// TIA Portal V17 export
// export: Created 2024-09-02T12:50:04.1377322Z, ExportSetting WithDefaults, DisplayName Totally Integrated Automation Portal, DisplayVersion V17, DisplayName TIA Portal Openness, DisplayVersion V17, DisplayName TIA Portal Version Control Interface, DisplayVersion V17, DisplayName STEP 7 Professional, DisplayVersion V17, DisplayName STEP 7 Safety, DisplayVersion V17, DisplayName WinCC Professional, DisplayVersion V17
FUNCTION_BLOCK "SysFB_RF300"   // FB809, LAD
TITLE = /RF300 Read / Write / RF300 Lesen / Schreiben
{ S7_Optimized_Access := 'TRUE' }
AUTHOR : STEAM
FAMILY : MOBY
NAME : MOBY
VERSION : 0.1
// stored: AutoNumber true, IsIECCheckEnabled false, IsRetainMemResEnabled false, MemoryReserve 100, SetENOAutomatically false, UDAEnableTagReadback false
   VAR_INPUT
      HW_ID : Int;   // Hardware ID
      HW_ADR : Int;   // Hardwareadresse / Hardware address
      Channel : Int;   // Kanalnummer (1..2) / Channel number (1..2)
      RF_Type : Bool;   // False=RF300 True= RF200
      "Fault ACK" : Bool;   // Fehler quittieren / Acknowledge error
      "New Start" : Bool;   // Flanke Neustart / Flank Restart
   END_VAR
   VAR_OUTPUT
      Fault : Bool;   // es ist ein Fehler aufgetreten / An error has occurred.
      "MDS Present" : Bool;   // Datenträger ist anwesend / Data carrier is present
      HMIDiag : "TypeMobyHMIDiag";   // HMI Diagnose / HMI Diagnosis
   END_VAR
   VAR_IN_OUT
      Command : "TypeMobyBefehle";
   END_VAR
   VAR
      hwConnect { S7_SetPoint := 'True'} : IID_HW_CONNECT;
      Reset : Struct
         Start : Bool;   // Start
         Active : Bool;   // Aktiv / Active
         Finish : Bool;   // Fertig / Finished
         Fault : Bool;   // Fehler / Error
         Status : DWord;   // Status
         Status_marked : DWord;   // Status
         Num_Of_OK : DInt;   // Anzahl IO / Number NIO
         Num_Of_NOK : DInt;   // Anzahl NIO / Number NIO
         started : Bool;   // Funktion gestartet / Function started
         fp_started : Bool;   // flanke gestartet / Flank started
         hm_fp_started : Bool;   // HM flanke gestartet / HM flank started
         Finish_OK : Bool;   // Fertig IO / Finish IO
         fp_Finish_OK : Bool;   // flanke Fertig IO / Flank finished OK
         "hm fp_Finish_OK" : Bool;   // hm flanke Fertig IO / hm flank finished IO
         Finish_NOK : Bool;   // Fertig NIO / Finish NIO
         fp_Finish_NOK : Bool;   // flanke Fertig IO / Flank finished OK
         "hm fp_Finish_NOK" : Bool;   // hm flanke Fertig IO / hm flank finished IO
         RunningTime : Time;
      END_STRUCT;
      Read : Struct
         Start : Bool;   // Start
         Active : Bool;   // Aktiv / Active
         Finish : Bool;   // Fertig / Finished
         Faul : Bool;   // Fehler / Error
         MDS_present : Bool;   // Datenträger vorhanden / Data carrier available
         Status : DWord;   // Status
         Status_marked : DWord;   // Status
         Num_Of_OK : DInt;   // Anzahl IO / Number NIO
         Num_Of_NOK : DInt;   // Anzahl NIO / Number NIO
         started : Bool;   // Funktion gestartet / Function started
         fp_started : Bool;   // flanke gestartet / Flank started
         hm_fp_started : Bool;   // HM flanke gestartet / HM flank started
         Finish_OK : Bool;   // Fertig IO / Finish IO
         fp_Finish_OK : Bool;   // flanke Fertig IO / Flank finished OK
         "hm fp_Finish_OK" : Bool;   // hm flanke Fertig IO / hm flank finished IO
         Finish_NOK : Bool;   // Fertig NIO / Finish NIO
         fp_Finish_NOK : Bool;   // flanke Fertig IO / Flank finished OK
         "hm fp_Finish_NOK" : Bool;   // hm flanke Fertig IO / hm flank finished IO
         RunningTime : Time;
      END_STRUCT;
      Write : Struct
         Start : Bool;   // Start
         Active : Bool;   // Aktiv / Active
         Finish : Bool;   // Fertig / Finished
         Fault : Bool;   // Fehler / Error
         MDS_present : Bool;   // Datenträger vorhanden / Data carrier available
         Status : DWord;   // Status
         Status_marked : DWord;   // Status
         Num_Of_OK : DInt;   // Anzahl IO / Number NIO
         Num_Of_NOK : DInt;   // Anzahl NIO / Number NIO
         started : Bool;   // Funktion gestartet / Function started
         fp_started : Bool;   // flanke gestartet / Flank started
         hm_fp_started : Bool;   // HM flanke gestartet / HM flank started
         Finish_OK : Bool;   // Fertig IO / Finish IO
         fp_Finish_OK : Bool;   // flanke Fertig IO / Flank finished OK
         "hm fp_Finish_OK" : Bool;   // hm flanke Fertig IO / hm flank finished IO
         Finish_NOK : Bool;   // Fertig NIO / Finish NIO
         fp_Finish_NOK : Bool;   // flanke Fertig IO / Flank finished OK
         "hm fp_Finish_NOK" : Bool;   // hm flanke Fertig IO / hm flank finished IO
         RunningTime : Time;
      END_STRUCT;
      SysDI_Reset { S7_SetPoint := 'True'} : Reset_RF300;
      SysDI_Read { S7_SetPoint := 'True'} : Read;
      SysDI_Write { S7_SetPoint := 'True'} : Write;
      SystemTime : Time;
      SystemTime_Old : Time;
      CycleTime : Time;
      ReadData : Struct
         SequenceNr : Int;
         RetVal : Word;
         Pos : DInt;
         finish : Bool;
      END_STRUCT;
      WriteData : Struct
         SequenceNr : Int;
         RetVal : Word;
         Pos : DInt;
         finish : Bool;
      END_STRUCT;
      ConnectionCheck : Struct
         TimeWithoutAction : Time;
         start : Bool;
         fp_start : Bool;
         HM_fp_start : Bool;
      END_STRUCT;
      "Checking Faults" : Struct
         FaultOccured : Bool;
         fp_FaultOccured : Bool;
         HM_fp_FaultOccured : Bool;
         TimeoutFault : Bool;
      END_STRUCT;
      SysDI_Reset200 { S7_SetPoint := 'True'} : Reset_RF200;
   END_VAR
   VAR_TEMP
      t_VKE0 : Bool;
      t_VKE1 : Bool;
      t_End : Bool;
      t_RF300_Ready : Bool;
      t_Befehl_INIT : "TypeMobySequenz";
   END_VAR
   VAR_TEMP   // added for the SCL form of the ladder/FBD networks
      _w1 : Bool;
      _w2 : Bool;
      _w3 : Bool;
   END_VAR
BEGIN

REGION Network 1: INIT
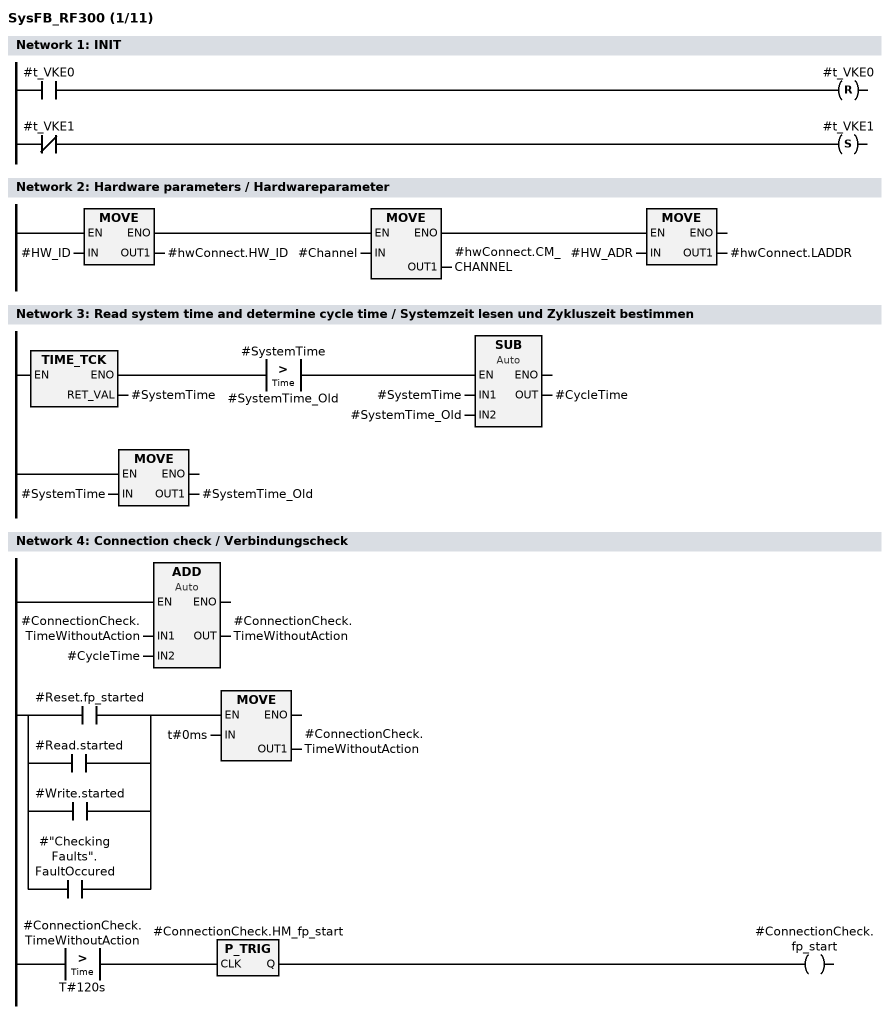
   RUNG wire#powerrail
      Contact( #t_VKE0 )
      R_Coil( #t_VKE0 )
   END_RUNG
   RUNG wire#powerrail
      I_Contact( #t_VKE1 )
      S_Coil( #t_VKE1 )
   END_RUNG
   // the same network as SCL:
   IF #t_VKE0 THEN #t_VKE0 := FALSE; END_IF;
   IF NOT #t_VKE1 THEN #t_VKE1 := TRUE; END_IF;
END_REGION

REGION Network 2: Hardware parameters / Hardwareparameter
   RUNG wire#powerrail
      Move(in := #HW_ID, out1 => #hwConnect.HW_ID)
      Move(in := #Channel, out1 => #hwConnect.CM_CHANNEL)
      Move(in := #HW_ADR, out1 => #hwConnect.LADDR)
   END_RUNG
   // the same network as SCL:
   #hwConnect.HW_ID := #HW_ID;
   #hwConnect.CM_CHANNEL := #Channel;
   #hwConnect.LADDR := #HW_ADR;
END_REGION

REGION Network 3: Read system time and determine cycle time / Systemzeit lesen und Zykluszeit bestimmen
   RUNG wire#powerrail
      TIME_TCK(RET_VAL => #SystemTime)
      { S7_Templates := "SrcType := Time" } GT_Contact(in1 := #SystemTime, in2 := #SystemTime_Old)
      Sub(in1 := #SystemTime, in2 := #SystemTime_Old, out => #CycleTime)
   END_RUNG
   RUNG wire#powerrail
      Move(in := #SystemTime, out1 => #SystemTime_Old)
   END_RUNG
   // the same network as SCL:
   #SystemTime := TIME_TCK(ENO => #_w1);
   IF #_w1 AND (#SystemTime > #SystemTime_Old) THEN #CycleTime := #SystemTime - #SystemTime_Old; END_IF;
   #SystemTime_Old := #SystemTime;
END_REGION

REGION Network 4: Connection check / Verbindungscheck
   RUNG wire#powerrail
      Add(in1 := #ConnectionCheck.TimeWithoutAction, in2 := #CycleTime, out => #ConnectionCheck.TimeWithoutAction)
   END_RUNG
   RUNG wire#powerrail
      Contact( #Reset.fp_started )
      wire#w1
      Move(in := t#0ms, out1 => #ConnectionCheck.TimeWithoutAction)
   END_RUNG
   RUNG wire#powerrail
      Contact( #Read.started )
   END_RUNG wire#w1
   RUNG wire#powerrail
      Contact( #Write.started )
   END_RUNG wire#w1
   RUNG wire#powerrail
      Contact( #"Checking Faults".FaultOccured )
   END_RUNG wire#w1
   RUNG wire#powerrail
      { S7_Templates := "SrcType := Time" } GT_Contact(in1 := #ConnectionCheck.TimeWithoutAction, in2 := T#120s)
      P_Trig( #ConnectionCheck.HM_fp_start )
      Coil( #ConnectionCheck.fp_start )
   END_RUNG
   // the same network as SCL:
   #ConnectionCheck.TimeWithoutAction := #ConnectionCheck.TimeWithoutAction + #CycleTime;
   IF #Reset.fp_started OR #Read.started OR #Write.started OR #"Checking Faults".FaultOccured THEN
       #ConnectionCheck.TimeWithoutAction := t#0ms;
   END_IF;
   #_w1 := #ConnectionCheck.TimeWithoutAction > T#120s;
   #_w2 := #_w1 AND NOT #ConnectionCheck.HM_fp_start;   // rising edge
   #ConnectionCheck.HM_fp_start := #_w1;
   #ConnectionCheck.fp_start := #_w2;
END_REGION

REGION Network 5: Error present / Fehler vorhanden
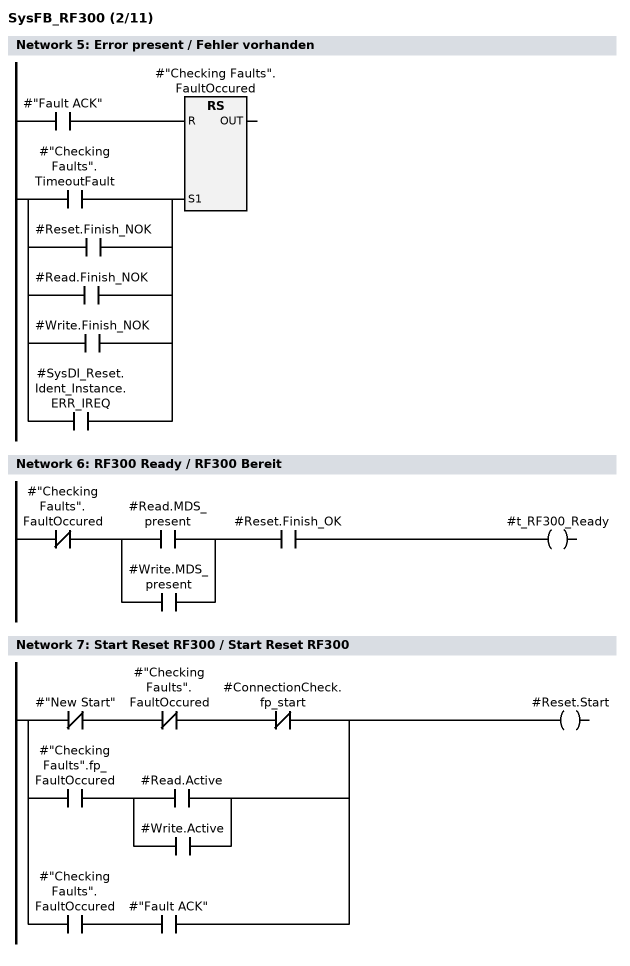
   RUNG wire#powerrail
      Contact( #"Fault ACK" )
      S_RS(operand := #"Checking Faults".FaultOccured, s1 := wire#w1)
   END_RUNG
   RUNG wire#powerrail
      Contact( #"Checking Faults".TimeoutFault )
   END_RUNG wire#w1
   RUNG wire#powerrail
      Contact( #Reset.Finish_NOK )
   END_RUNG wire#w1
   RUNG wire#powerrail
      Contact( #Read.Finish_NOK )
   END_RUNG wire#w1
   RUNG wire#powerrail
      Contact( #Write.Finish_NOK )
   END_RUNG wire#w1
   RUNG wire#powerrail
      Contact( #SysDI_Reset.Ident_Instance.ERR_IREQ )
   END_RUNG wire#w1
   // the same network as SCL:
   IF #"Fault ACK" THEN
       #"Checking Faults".FaultOccured := FALSE;   // RS flip-flop
   END_IF;
   IF #"Checking Faults".TimeoutFault OR #Reset.Finish_NOK OR #Read.Finish_NOK OR #Write.Finish_NOK OR #SysDI_Reset.Ident_Instance.ERR_IREQ THEN
       #"Checking Faults".FaultOccured := TRUE;
   END_IF;
END_REGION

REGION Network 6: RF300 Ready / RF300 Bereit
   RUNG wire#powerrail
      I_Contact( #"Checking Faults".FaultOccured )
      wire#w1
      Contact( #Read.MDS_present )
      wire#w2
      Contact( #Reset.Finish_OK )
      Coil( #t_RF300_Ready )
   END_RUNG
   RUNG wire#w1
      Contact( #Write.MDS_present )
   END_RUNG wire#w2
   // the same network as SCL:
   #t_RF300_Ready := NOT #"Checking Faults".FaultOccured AND (#Read.MDS_present OR #Write.MDS_present) AND #Reset.Finish_OK;
END_REGION

REGION Network 7: Start Reset RF300 / Start Reset RF300
   RUNG wire#powerrail
      I_Contact( #"New Start" )
      I_Contact( #"Checking Faults".FaultOccured )
      I_Contact( #ConnectionCheck.fp_start )
      wire#w1
      Coil( #Reset.Start )
   END_RUNG
   RUNG wire#powerrail
      Contact( #"Checking Faults".fp_FaultOccured )
      wire#w2
      Contact( #Read.Active )
   END_RUNG wire#w1
   RUNG wire#w2
      Contact( #Write.Active )
   END_RUNG wire#w1
   RUNG wire#powerrail
      Contact( #"Checking Faults".FaultOccured )
      Contact( #"Fault ACK" )
   END_RUNG wire#w1
   // the same network as SCL:
   #Reset.Start := (NOT #"New Start" AND NOT #"Checking Faults".FaultOccured AND NOT #ConnectionCheck.fp_start) OR (#"Checking Faults".fp_FaultOccured AND (#Read.Active OR #Write.Active)) OR (#"Checking Faults".FaultOccured AND #"Fault ACK");
END_REGION

REGION Network 8: Reset RF300
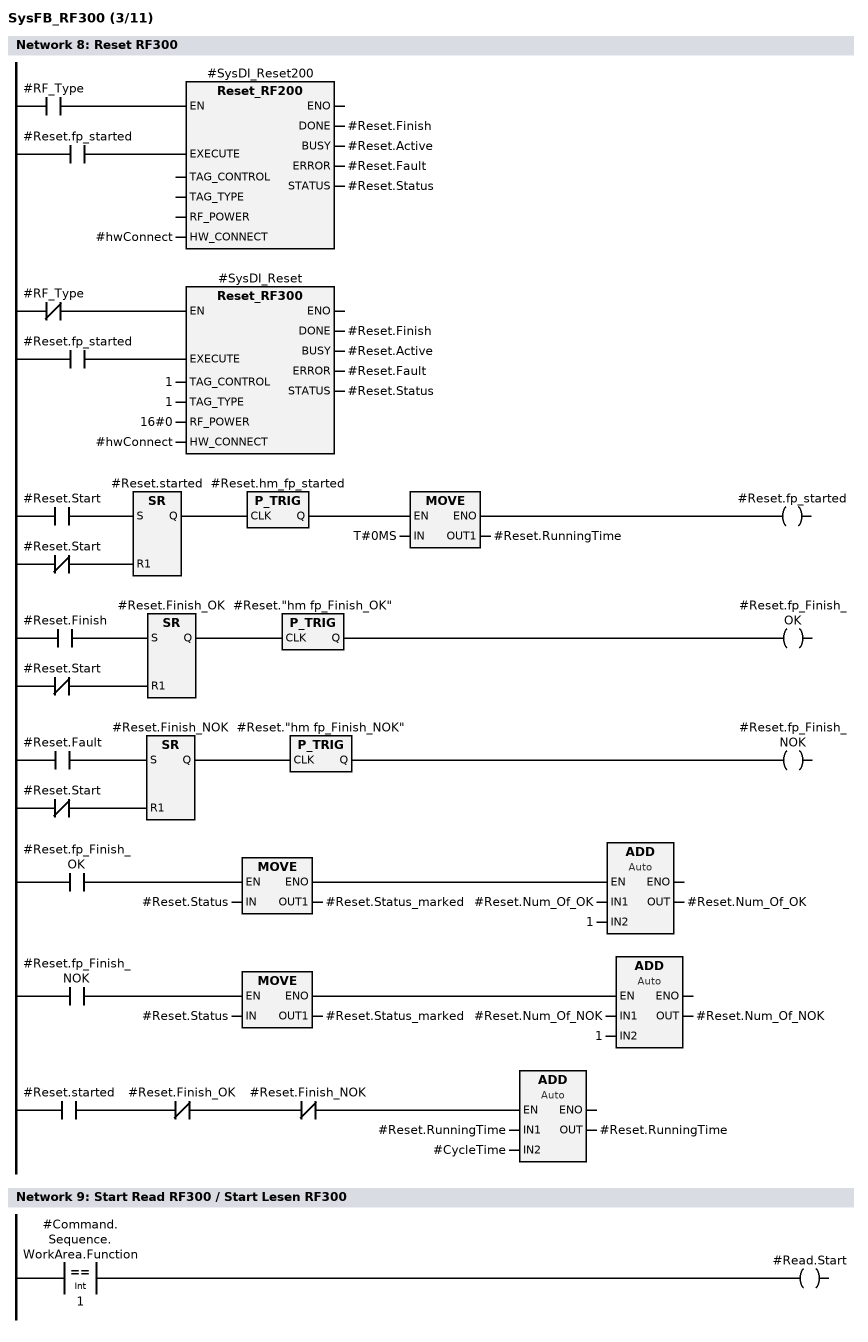
   RUNG wire#powerrail
      Contact( #RF_Type )
      #SysDI_Reset200.Reset_RF200(EXECUTE := wire#w1, TAG_CONTROL :=, TAG_TYPE :=, RF_POWER :=, HW_CONNECT := #hwConnect, DONE => #Reset.Finish, BUSY => #Reset.Active, ERROR => #Reset.Fault, STATUS => #Reset.Status)
   END_RUNG
   RUNG wire#powerrail
      Contact( #Reset.fp_started )
   END_RUNG wire#w1
   RUNG wire#powerrail
      I_Contact( #RF_Type )
      #SysDI_Reset.Reset_RF300(EXECUTE := wire#w2, TAG_CONTROL := 1, TAG_TYPE := 1, RF_POWER := 16#0, HW_CONNECT := #hwConnect, DONE => #Reset.Finish, BUSY => #Reset.Active, ERROR => #Reset.Fault, STATUS => #Reset.Status)
   END_RUNG
   RUNG wire#powerrail
      Contact( #Reset.fp_started )
   END_RUNG wire#w2
   RUNG wire#powerrail
      Contact( #Reset.Start )
      S_SR(operand := #Reset.started, r1 := wire#w3)
      P_Trig( #Reset.hm_fp_started )
      Move(in := T#0MS, out1 => #Reset.RunningTime)
      Coil( #Reset.fp_started )
   END_RUNG
   RUNG wire#powerrail
      I_Contact( #Reset.Start )
   END_RUNG wire#w3
   RUNG wire#powerrail
      Contact( #Reset.Finish )
      S_SR(operand := #Reset.Finish_OK, r1 := wire#w4)
      P_Trig( #Reset."hm fp_Finish_OK" )
      Coil( #Reset.fp_Finish_OK )
   END_RUNG
   RUNG wire#powerrail
      I_Contact( #Reset.Start )
   END_RUNG wire#w4
   RUNG wire#powerrail
      Contact( #Reset.Fault )
      S_SR(operand := #Reset.Finish_NOK, r1 := wire#w5)
      P_Trig( #Reset."hm fp_Finish_NOK" )
      Coil( #Reset.fp_Finish_NOK )
   END_RUNG
   RUNG wire#powerrail
      I_Contact( #Reset.Start )
   END_RUNG wire#w5
   RUNG wire#powerrail
      Contact( #Reset.fp_Finish_OK )
      Move(in := #Reset.Status, out1 => #Reset.Status_marked)
      Add(in1 := #Reset.Num_Of_OK, in2 := 1, out => #Reset.Num_Of_OK)
   END_RUNG
   RUNG wire#powerrail
      Contact( #Reset.fp_Finish_NOK )
      Move(in := #Reset.Status, out1 => #Reset.Status_marked)
      Add(in1 := #Reset.Num_Of_NOK, in2 := 1, out => #Reset.Num_Of_NOK)
   END_RUNG
   RUNG wire#powerrail
      Contact( #Reset.started )
      I_Contact( #Reset.Finish_OK )
      I_Contact( #Reset.Finish_NOK )
      Add(in1 := #Reset.RunningTime, in2 := #CycleTime, out => #Reset.RunningTime)
   END_RUNG
   // the same network as SCL:
   IF #RF_Type THEN
       #SysDI_Reset200(EXECUTE := #Reset.fp_started,   // Reset_RF200
                       HW_CONNECT := #hwConnect,
                       DONE => #Reset.Finish,
                       BUSY => #Reset.Active,
                       ERROR => #Reset.Fault,
                       STATUS => #Reset.Status);
   END_IF;
   IF NOT #RF_Type THEN
       #SysDI_Reset(EXECUTE := #Reset.fp_started,   // Reset_RF300
                    TAG_CONTROL := 1,
                    TAG_TYPE := 1,
                    RF_POWER := 16#0,
                    HW_CONNECT := #hwConnect,
                    DONE => #Reset.Finish,
                    BUSY => #Reset.Active,
                    ERROR => #Reset.Fault,
                    STATUS => #Reset.Status);
   END_IF;
   IF #Reset.Start THEN
       #Reset.started := TRUE;   // SR flip-flop
   END_IF;
   IF NOT #Reset.Start THEN #Reset.started := FALSE; END_IF;
   #_w1 := #Reset.started AND NOT #Reset.hm_fp_started;   // rising edge
   #Reset.hm_fp_started := #Reset.started;
   IF #_w1 THEN #Reset.RunningTime := T#0MS; END_IF;
   #Reset.fp_started := #_w1;
   IF #Reset.Finish THEN
       #Reset.Finish_OK := TRUE;   // SR flip-flop
   END_IF;
   IF NOT #Reset.Start THEN #Reset.Finish_OK := FALSE; END_IF;
   #_w2 := #Reset.Finish_OK AND NOT #Reset."hm fp_Finish_OK";   // rising edge
   #Reset."hm fp_Finish_OK" := #Reset.Finish_OK;
   #Reset.fp_Finish_OK := #_w2;
   IF #Reset.Fault THEN
       #Reset.Finish_NOK := TRUE;   // SR flip-flop
   END_IF;
   IF NOT #Reset.Start THEN #Reset.Finish_NOK := FALSE; END_IF;
   #_w3 := #Reset.Finish_NOK AND NOT #Reset."hm fp_Finish_NOK";   // rising edge
   #Reset."hm fp_Finish_NOK" := #Reset.Finish_NOK;
   #Reset.fp_Finish_NOK := #_w3;
   IF #Reset.fp_Finish_OK THEN
       #Reset.Status_marked := #Reset.Status;
       #Reset.Num_Of_OK := #Reset.Num_Of_OK + 1;
   END_IF;
   IF #Reset.fp_Finish_NOK THEN
       #Reset.Status_marked := #Reset.Status;
       #Reset.Num_Of_NOK := #Reset.Num_Of_NOK + 1;
   END_IF;
   IF #Reset.started AND NOT #Reset.Finish_OK AND NOT #Reset.Finish_NOK THEN
       #Reset.RunningTime := #Reset.RunningTime + #CycleTime;
   END_IF;
END_REGION

REGION Network 9: Start Read RF300 / Start Lesen RF300
   RUNG wire#powerrail
      { S7_Templates := "SrcType := Int" } EQ_Contact(in1 := #Command.Sequence.WorkArea.Function, in2 := 1)
      Coil( #Read.Start )
   END_RUNG
   // the same network as SCL:
   #Read.Start := #Command.Sequence.WorkArea.Function = 1;
END_REGION

REGION Network 10: Read RF300 / Lesen RF300
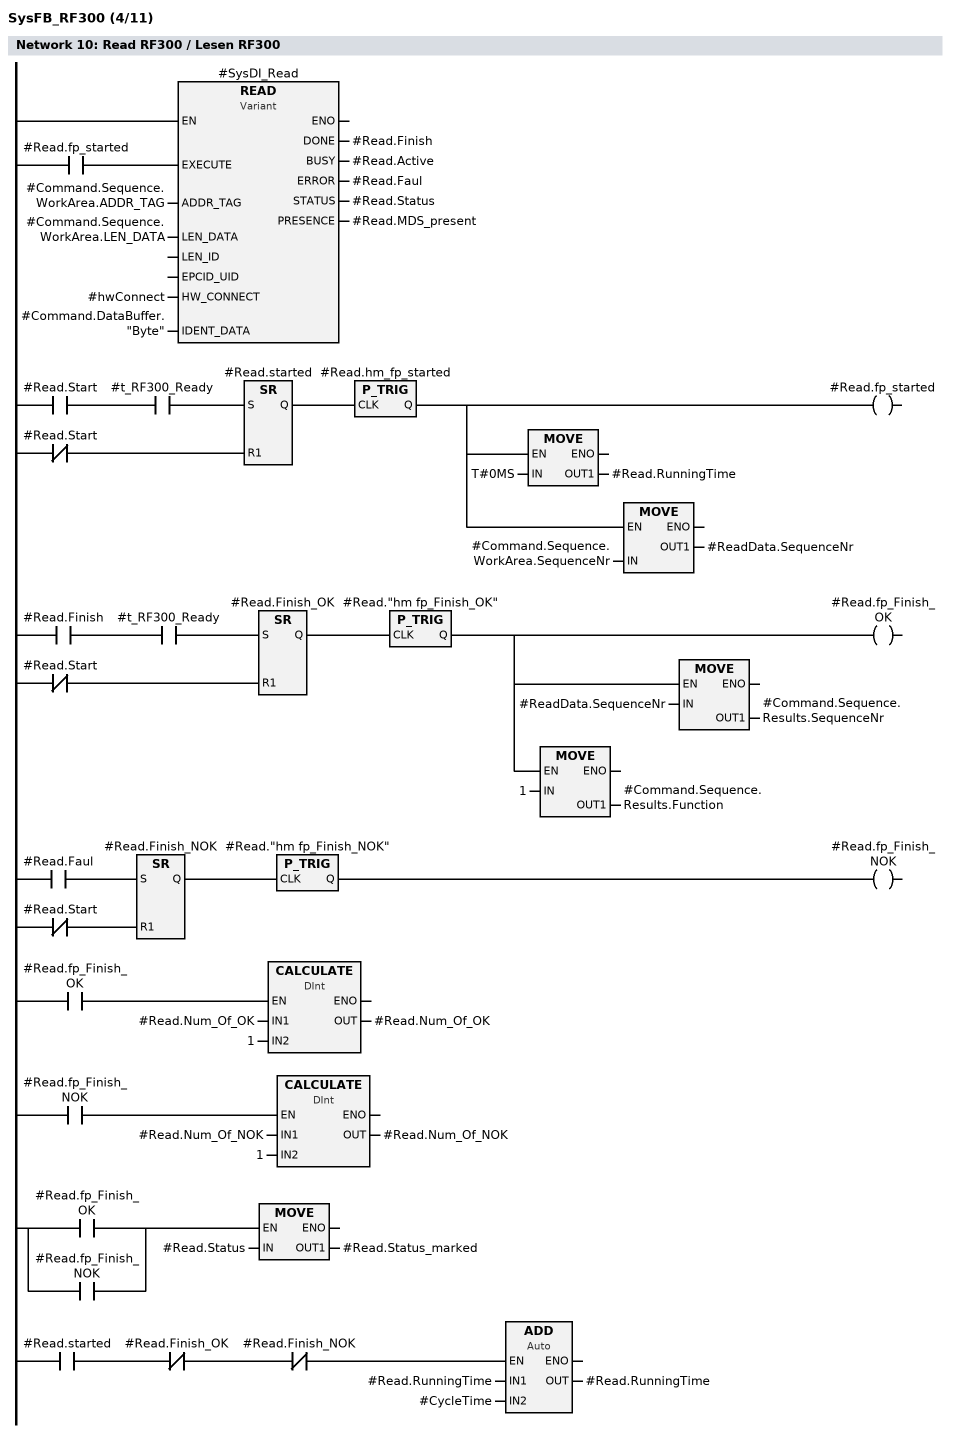
   RUNG wire#powerrail
      { S7_Templates := "ident_data_type := Variant" } #SysDI_Read.Read(EXECUTE := wire#w1, ADDR_TAG := #Command.Sequence.WorkArea.ADDR_TAG, LEN_DATA := #Command.Sequence.WorkArea.LEN_DATA, LEN_ID :=, EPCID_UID :=, HW_CONNECT := #hwConnect, IDENT_DATA := #Command.DataBuffer."Byte", DONE => #Read.Finish, BUSY => #Read.Active, ERROR => #Read.Faul, STATUS => #Read.Status, PRESENCE => #Read.MDS_present)
   END_RUNG
   RUNG wire#powerrail
      Contact( #Read.fp_started )
   END_RUNG wire#w1
   RUNG wire#powerrail
      Contact( #Read.Start )
      Contact( #t_RF300_Ready )
      S_SR(operand := #Read.started, r1 := wire#w2)
      P_Trig( #Read.hm_fp_started )
      wire#w3
      Coil( #Read.fp_started )
   END_RUNG
   RUNG wire#powerrail
      I_Contact( #Read.Start )
   END_RUNG wire#w2
   RUNG wire#w3
      Move(in := T#0MS, out1 => #Read.RunningTime)
   END_RUNG
   RUNG wire#w3
      Move(in := #Command.Sequence.WorkArea.SequenceNr, out1 => #ReadData.SequenceNr)
   END_RUNG
   RUNG wire#powerrail
      Contact( #Read.Finish )
      Contact( #t_RF300_Ready )
      S_SR(operand := #Read.Finish_OK, r1 := wire#w4)
      P_Trig( #Read."hm fp_Finish_OK" )
      wire#w5
      Coil( #Read.fp_Finish_OK )
   END_RUNG
   RUNG wire#powerrail
      I_Contact( #Read.Start )
   END_RUNG wire#w4
   RUNG wire#w5
      Move(in := #ReadData.SequenceNr, out1 => #Command.Sequence.Results.SequenceNr)
   END_RUNG
   RUNG wire#w5
      Move(in := 1, out1 => #Command.Sequence.Results.Function)
   END_RUNG
   RUNG wire#powerrail
      Contact( #Read.Faul )
      S_SR(operand := #Read.Finish_NOK, r1 := wire#w6)
      P_Trig( #Read."hm fp_Finish_NOK" )
      Coil( #Read.fp_Finish_NOK )
   END_RUNG
   RUNG wire#powerrail
      I_Contact( #Read.Start )
   END_RUNG wire#w6
   RUNG wire#powerrail
      Contact( #Read.fp_Finish_OK )
      { S7_Templates := "SrcType := DInt"; S7_Expression := "IN1+IN2" } Calculate(in1 := #Read.Num_Of_OK, in2 := 1, out => #Read.Num_Of_OK)
   END_RUNG
   RUNG wire#powerrail
      Contact( #Read.fp_Finish_NOK )
      { S7_Templates := "SrcType := DInt"; S7_Expression := "IN1+IN2" } Calculate(in1 := #Read.Num_Of_NOK, in2 := 1, out => #Read.Num_Of_NOK)
   END_RUNG
   RUNG wire#powerrail
      Contact( #Read.fp_Finish_OK )
      wire#w7
      Move(in := #Read.Status, out1 => #Read.Status_marked)
   END_RUNG
   RUNG wire#powerrail
      Contact( #Read.fp_Finish_NOK )
   END_RUNG wire#w7
   RUNG wire#powerrail
      Contact( #Read.started )
      I_Contact( #Read.Finish_OK )
      I_Contact( #Read.Finish_NOK )
      Add(in1 := #Read.RunningTime, in2 := #CycleTime, out => #Read.RunningTime)
   END_RUNG
   // the same network as SCL:
   #SysDI_Read(EXECUTE := #Read.fp_started,   // Read
               ADDR_TAG := #Command.Sequence.WorkArea.ADDR_TAG,
               LEN_DATA := #Command.Sequence.WorkArea.LEN_DATA,
               HW_CONNECT := #hwConnect,
               IDENT_DATA := #Command.DataBuffer."Byte",
               DONE => #Read.Finish,
               BUSY => #Read.Active,
               ERROR => #Read.Faul,
               STATUS => #Read.Status,
               PRESENCE => #Read.MDS_present);
   IF #Read.Start AND #t_RF300_Ready THEN
       #Read.started := TRUE;   // SR flip-flop
   END_IF;
   IF NOT #Read.Start THEN #Read.started := FALSE; END_IF;
   #_w1 := #Read.started AND NOT #Read.hm_fp_started;   // rising edge
   #Read.hm_fp_started := #Read.started;
   #Read.fp_started := #_w1;
   IF #_w1 THEN
       #Read.RunningTime := T#0MS;
       #ReadData.SequenceNr := #Command.Sequence.WorkArea.SequenceNr;
   END_IF;
   IF #Read.Finish AND #t_RF300_Ready THEN
       #Read.Finish_OK := TRUE;   // SR flip-flop
   END_IF;
   IF NOT #Read.Start THEN #Read.Finish_OK := FALSE; END_IF;
   #_w2 := #Read.Finish_OK AND NOT #Read."hm fp_Finish_OK";   // rising edge
   #Read."hm fp_Finish_OK" := #Read.Finish_OK;
   #Read.fp_Finish_OK := #_w2;
   IF #_w2 THEN
       #Command.Sequence.Results.SequenceNr := #ReadData.SequenceNr;
       #Command.Sequence.Results.Function := 1;
   END_IF;
   IF #Read.Faul THEN
       #Read.Finish_NOK := TRUE;   // SR flip-flop
   END_IF;
   IF NOT #Read.Start THEN #Read.Finish_NOK := FALSE; END_IF;
   #_w3 := #Read.Finish_NOK AND NOT #Read."hm fp_Finish_NOK";   // rising edge
   #Read."hm fp_Finish_NOK" := #Read.Finish_NOK;
   #Read.fp_Finish_NOK := #_w3;
   IF #Read.fp_Finish_OK THEN #Read.Num_Of_OK := #Read.Num_Of_OK+1; END_IF;
   IF #Read.fp_Finish_NOK THEN #Read.Num_Of_NOK := #Read.Num_Of_NOK+1; END_IF;
   IF #Read.fp_Finish_OK OR #Read.fp_Finish_NOK THEN #Read.Status_marked := #Read.Status; END_IF;
   IF #Read.started AND NOT #Read.Finish_OK AND NOT #Read.Finish_NOK THEN
       #Read.RunningTime := #Read.RunningTime + #CycleTime;
   END_IF;
END_REGION

REGION Network 11: Start writing RF300 / Start Schreiben RF300
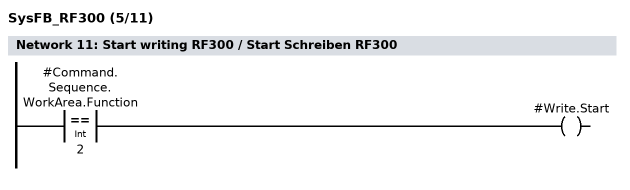
   RUNG wire#powerrail
      { S7_Templates := "SrcType := Int" } EQ_Contact(in1 := #Command.Sequence.WorkArea.Function, in2 := 2)
      Coil( #Write.Start )
   END_RUNG
   // the same network as SCL:
   #Write.Start := #Command.Sequence.WorkArea.Function = 2;
END_REGION

REGION Network 12: Write RF300 / Schreiben RF300
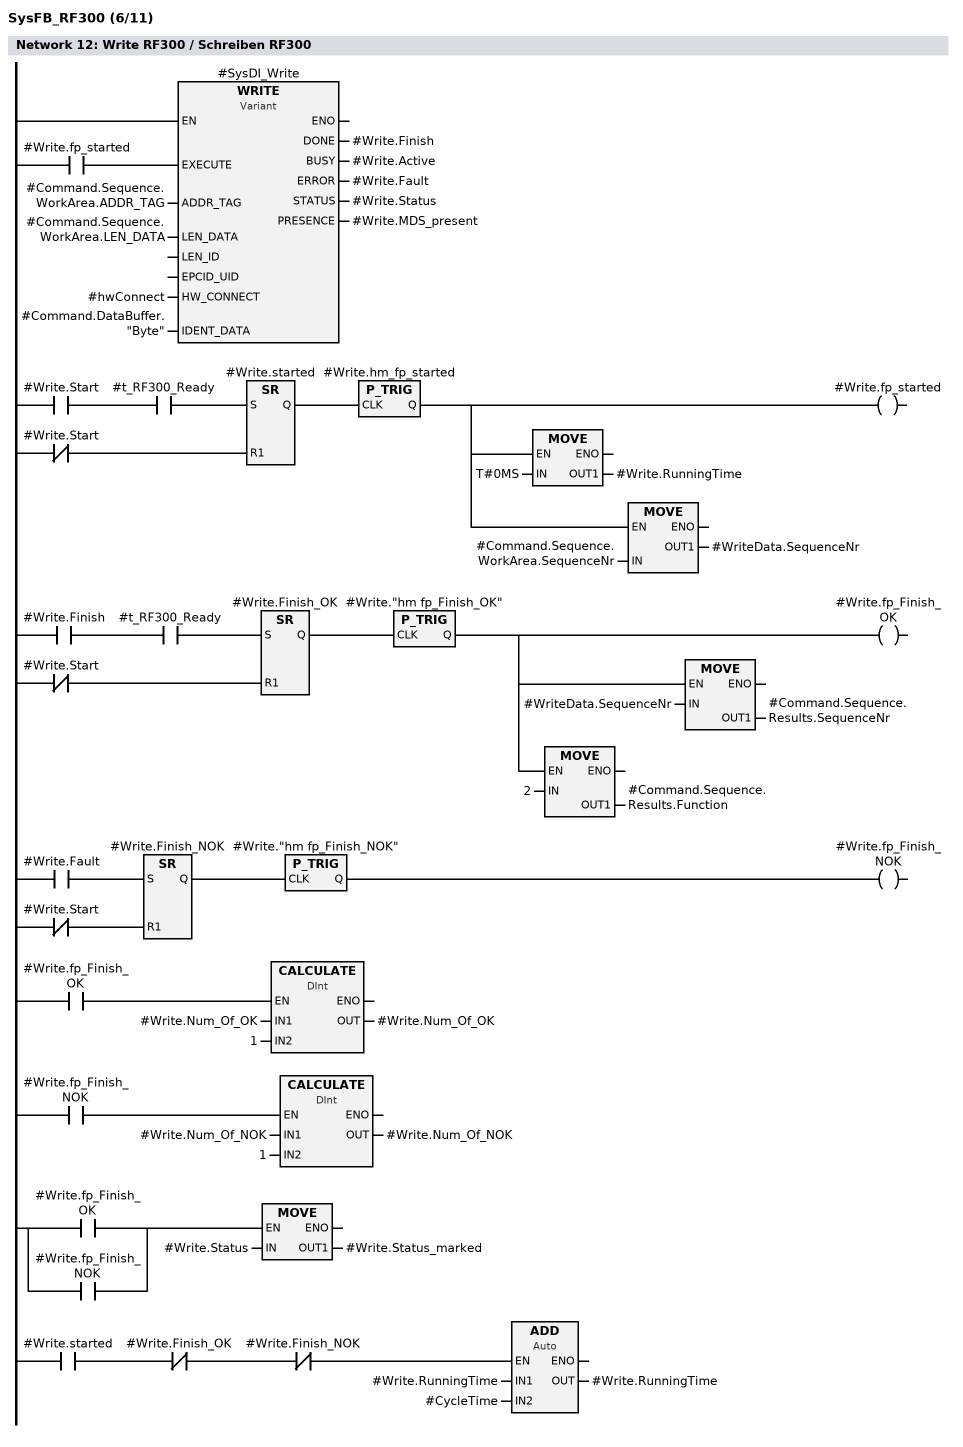
   RUNG wire#powerrail
      { S7_Templates := "ident_data_type := Variant" } #SysDI_Write.Write(EXECUTE := wire#w1, ADDR_TAG := #Command.Sequence.WorkArea.ADDR_TAG, LEN_DATA := #Command.Sequence.WorkArea.LEN_DATA, LEN_ID :=, EPCID_UID :=, HW_CONNECT := #hwConnect, IDENT_DATA := #Command.DataBuffer."Byte", DONE => #Write.Finish, BUSY => #Write.Active, ERROR => #Write.Fault, STATUS => #Write.Status, PRESENCE => #Write.MDS_present)
   END_RUNG
   RUNG wire#powerrail
      Contact( #Write.fp_started )
   END_RUNG wire#w1
   RUNG wire#powerrail
      Contact( #Write.Start )
      Contact( #t_RF300_Ready )
      S_SR(operand := #Write.started, r1 := wire#w2)
      P_Trig( #Write.hm_fp_started )
      wire#w3
      Coil( #Write.fp_started )
   END_RUNG
   RUNG wire#powerrail
      I_Contact( #Write.Start )
   END_RUNG wire#w2
   RUNG wire#w3
      Move(in := T#0MS, out1 => #Write.RunningTime)
   END_RUNG
   RUNG wire#w3
      Move(in := #Command.Sequence.WorkArea.SequenceNr, out1 => #WriteData.SequenceNr)
   END_RUNG
   RUNG wire#powerrail
      Contact( #Write.Finish )
      Contact( #t_RF300_Ready )
      S_SR(operand := #Write.Finish_OK, r1 := wire#w4)
      P_Trig( #Write."hm fp_Finish_OK" )
      wire#w5
      Coil( #Write.fp_Finish_OK )
   END_RUNG
   RUNG wire#powerrail
      I_Contact( #Write.Start )
   END_RUNG wire#w4
   RUNG wire#w5
      Move(in := #WriteData.SequenceNr, out1 => #Command.Sequence.Results.SequenceNr)
   END_RUNG
   RUNG wire#w5
      Move(in := 2, out1 => #Command.Sequence.Results.Function)
   END_RUNG
   RUNG wire#powerrail
      Contact( #Write.Fault )
      S_SR(operand := #Write.Finish_NOK, r1 := wire#w6)
      P_Trig( #Write."hm fp_Finish_NOK" )
      Coil( #Write.fp_Finish_NOK )
   END_RUNG
   RUNG wire#powerrail
      I_Contact( #Write.Start )
   END_RUNG wire#w6
   RUNG wire#powerrail
      Contact( #Write.fp_Finish_OK )
      { S7_Templates := "SrcType := DInt"; S7_Expression := "IN1+IN2" } Calculate(in1 := #Write.Num_Of_OK, in2 := 1, out => #Write.Num_Of_OK)
   END_RUNG
   RUNG wire#powerrail
      Contact( #Write.fp_Finish_NOK )
      { S7_Templates := "SrcType := DInt"; S7_Expression := "IN1+IN2" } Calculate(in1 := #Write.Num_Of_NOK, in2 := 1, out => #Write.Num_Of_NOK)
   END_RUNG
   RUNG wire#powerrail
      Contact( #Write.fp_Finish_OK )
      wire#w7
      Move(in := #Write.Status, out1 => #Write.Status_marked)
   END_RUNG
   RUNG wire#powerrail
      Contact( #Write.fp_Finish_NOK )
   END_RUNG wire#w7
   RUNG wire#powerrail
      Contact( #Write.started )
      I_Contact( #Write.Finish_OK )
      I_Contact( #Write.Finish_NOK )
      Add(in1 := #Write.RunningTime, in2 := #CycleTime, out => #Write.RunningTime)
   END_RUNG
   // the same network as SCL:
   #SysDI_Write(EXECUTE := #Write.fp_started,   // Write
                ADDR_TAG := #Command.Sequence.WorkArea.ADDR_TAG,
                LEN_DATA := #Command.Sequence.WorkArea.LEN_DATA,
                HW_CONNECT := #hwConnect,
                IDENT_DATA := #Command.DataBuffer."Byte",
                DONE => #Write.Finish,
                BUSY => #Write.Active,
                ERROR => #Write.Fault,
                STATUS => #Write.Status,
                PRESENCE => #Write.MDS_present);
   IF #Write.Start AND #t_RF300_Ready THEN
       #Write.started := TRUE;   // SR flip-flop
   END_IF;
   IF NOT #Write.Start THEN #Write.started := FALSE; END_IF;
   #_w1 := #Write.started AND NOT #Write.hm_fp_started;   // rising edge
   #Write.hm_fp_started := #Write.started;
   #Write.fp_started := #_w1;
   IF #_w1 THEN
       #Write.RunningTime := T#0MS;
       #WriteData.SequenceNr := #Command.Sequence.WorkArea.SequenceNr;
   END_IF;
   IF #Write.Finish AND #t_RF300_Ready THEN
       #Write.Finish_OK := TRUE;   // SR flip-flop
   END_IF;
   IF NOT #Write.Start THEN #Write.Finish_OK := FALSE; END_IF;
   #_w2 := #Write.Finish_OK AND NOT #Write."hm fp_Finish_OK";   // rising edge
   #Write."hm fp_Finish_OK" := #Write.Finish_OK;
   #Write.fp_Finish_OK := #_w2;
   IF #_w2 THEN
       #Command.Sequence.Results.SequenceNr := #WriteData.SequenceNr;
       #Command.Sequence.Results.Function := 2;
   END_IF;
   IF #Write.Fault THEN
       #Write.Finish_NOK := TRUE;   // SR flip-flop
   END_IF;
   IF NOT #Write.Start THEN #Write.Finish_NOK := FALSE; END_IF;
   #_w3 := #Write.Finish_NOK AND NOT #Write."hm fp_Finish_NOK";   // rising edge
   #Write."hm fp_Finish_NOK" := #Write.Finish_NOK;
   #Write.fp_Finish_NOK := #_w3;
   IF #Write.fp_Finish_OK THEN #Write.Num_Of_OK := #Write.Num_Of_OK+1; END_IF;
   IF #Write.fp_Finish_NOK THEN #Write.Num_Of_NOK := #Write.Num_Of_NOK+1; END_IF;
   IF #Write.fp_Finish_OK OR #Write.fp_Finish_NOK THEN #Write.Status_marked := #Write.Status; END_IF;
   IF #Write.started AND NOT #Write.Finish_OK AND NOT #Write.Finish_NOK THEN
       #Write.RunningTime := #Write.RunningTime + #CycleTime;
   END_IF;
END_REGION

REGION Network 13: Delete order compartment / Auftragsfach ablöschen
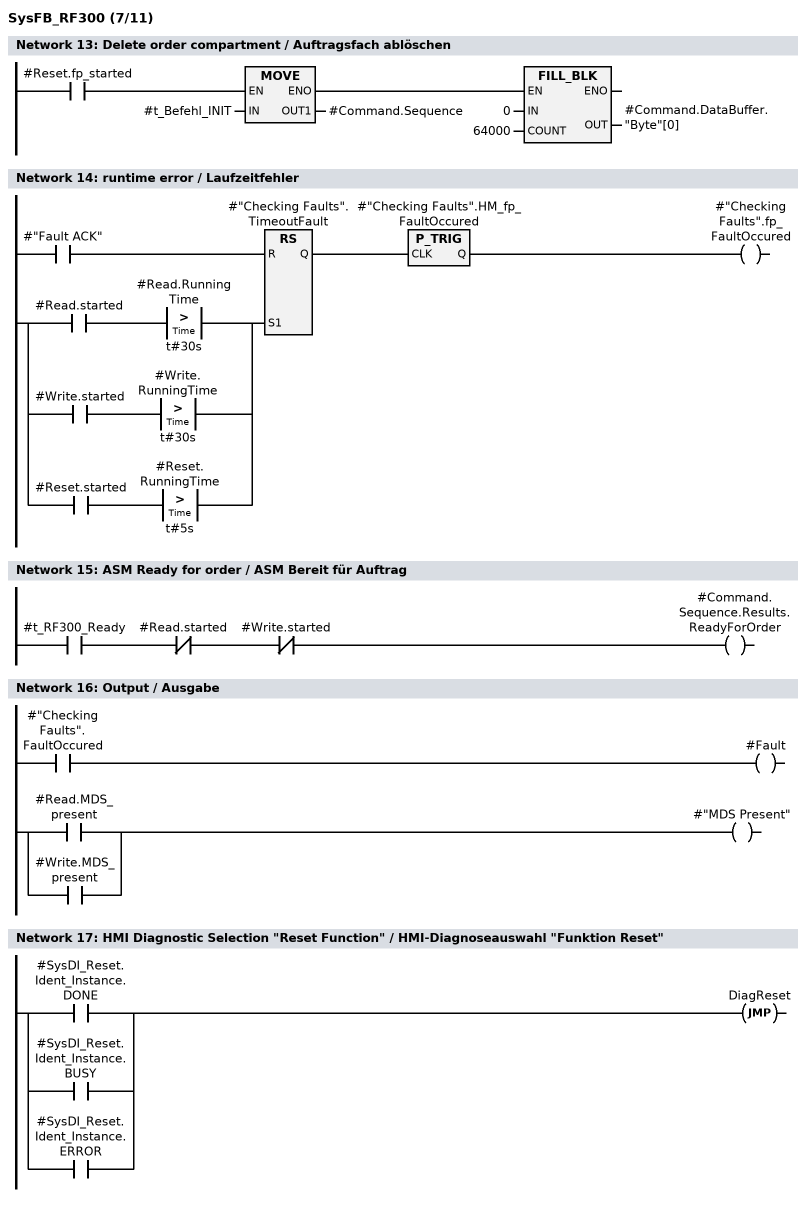
   RUNG wire#powerrail
      Contact( #Reset.fp_started )
      Move(in := #t_Befehl_INIT, out1 => #Command.Sequence)
      FillBlockI(in := 0, count := 64000, out => #Command.DataBuffer."Byte"[0])
   END_RUNG
   // the same network as SCL:
   IF #Reset.fp_started THEN
       #Command.Sequence := #t_Befehl_INIT;
       FILL_BLK(IN := 0, COUNT := 64000, OUT => #Command.DataBuffer."Byte"[0]);
   END_IF;
END_REGION

REGION Network 14: runtime error / Laufzeitfehler
   RUNG wire#powerrail
      Contact( #"Fault ACK" )
      S_RS(operand := #"Checking Faults".TimeoutFault, s1 := wire#w1)
      P_Trig( #"Checking Faults".HM_fp_FaultOccured )
      Coil( #"Checking Faults".fp_FaultOccured )
   END_RUNG
   RUNG wire#powerrail
      Contact( #Read.started )
      { S7_Templates := "SrcType := Time" } GT_Contact(in1 := #Read.RunningTime, in2 := t#30s)
   END_RUNG wire#w1
   RUNG wire#powerrail
      Contact( #Write.started )
      { S7_Templates := "SrcType := Time" } GT_Contact(in1 := #Write.RunningTime, in2 := t#30s)
   END_RUNG wire#w1
   RUNG wire#powerrail
      Contact( #Reset.started )
      { S7_Templates := "SrcType := Time" } GT_Contact(in1 := #Reset.RunningTime, in2 := t#5s)
   END_RUNG wire#w1
   // the same network as SCL:
   IF #"Fault ACK" THEN
       #"Checking Faults".TimeoutFault := FALSE;   // RS flip-flop
   END_IF;
   IF (#Read.started AND (#Read.RunningTime > t#30s)) OR (#Write.started AND (#Write.RunningTime > t#30s)) OR (#Reset.started AND (#Reset.RunningTime > t#5s)) THEN
       #"Checking Faults".TimeoutFault := TRUE;
   END_IF;
   #_w1 := #"Checking Faults".TimeoutFault AND NOT #"Checking Faults".HM_fp_FaultOccured;   // rising edge
   #"Checking Faults".HM_fp_FaultOccured := #"Checking Faults".TimeoutFault;
   #"Checking Faults".fp_FaultOccured := #_w1;
END_REGION

REGION Network 15: ASM Ready for order / ASM Bereit für Auftrag
   RUNG wire#powerrail
      Contact( #t_RF300_Ready )
      I_Contact( #Read.started )
      I_Contact( #Write.started )
      Coil( #Command.Sequence.Results.ReadyForOrder )
   END_RUNG
   // the same network as SCL:
   #Command.Sequence.Results.ReadyForOrder := #t_RF300_Ready AND NOT #Read.started AND NOT #Write.started;
END_REGION

REGION Network 16: Output / Ausgabe
   RUNG wire#powerrail
      Contact( #"Checking Faults".FaultOccured )
      Coil( #Fault )
   END_RUNG
   RUNG wire#powerrail
      Contact( #Read.MDS_present )
      wire#w1
      Coil( #"MDS Present" )
   END_RUNG
   RUNG wire#powerrail
      Contact( #Write.MDS_present )
   END_RUNG wire#w1
   // the same network as SCL:
   #Fault := #"Checking Faults".FaultOccured;
   #"MDS Present" := #Read.MDS_present OR #Write.MDS_present;
END_REGION

REGION Network 17: HMI Diagnostic Selection "Reset Function" / HMI-Diagnoseauswahl "Funktion Reset"
   RUNG wire#powerrail
      Contact( #SysDI_Reset.Ident_Instance.DONE )
      wire#w1
      JumpCoil( DiagReset )
   END_RUNG
   RUNG wire#powerrail
      Contact( #SysDI_Reset.Ident_Instance.BUSY )
   END_RUNG wire#w1
   RUNG wire#powerrail
      Contact( #SysDI_Reset.Ident_Instance.ERROR )
   END_RUNG wire#w1
   // the same network as SCL:
   IF #SysDI_Reset.Ident_Instance.DONE OR #SysDI_Reset.Ident_Instance.BUSY OR #SysDI_Reset.Ident_Instance.ERROR THEN
       GOTO DiagReset;
   END_IF;
END_REGION

REGION Network 18: HMI Diagnosis Selection "Read Function" / HMI-Diagnoseauswahl "Funktion Lesen"
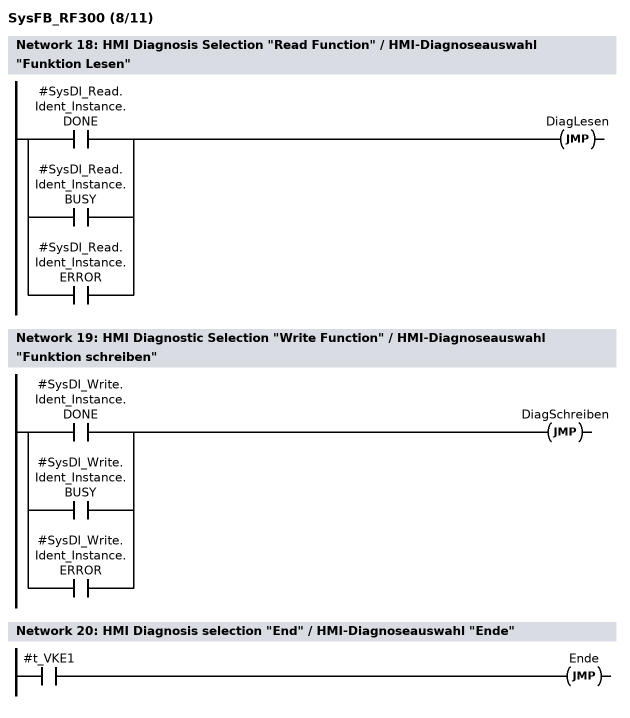
   RUNG wire#powerrail
      Contact( #SysDI_Read.Ident_Instance.DONE )
      wire#w1
      JumpCoil( DiagLesen )
   END_RUNG
   RUNG wire#powerrail
      Contact( #SysDI_Read.Ident_Instance.BUSY )
   END_RUNG wire#w1
   RUNG wire#powerrail
      Contact( #SysDI_Read.Ident_Instance.ERROR )
   END_RUNG wire#w1
   // the same network as SCL:
   IF #SysDI_Read.Ident_Instance.DONE OR #SysDI_Read.Ident_Instance.BUSY OR #SysDI_Read.Ident_Instance.ERROR THEN
       GOTO DiagLesen;
   END_IF;
END_REGION

REGION Network 19: HMI Diagnostic Selection "Write Function" / HMI-Diagnoseauswahl "Funktion schreiben"
   RUNG wire#powerrail
      Contact( #SysDI_Write.Ident_Instance.DONE )
      wire#w1
      JumpCoil( DiagSchreiben )
   END_RUNG
   RUNG wire#powerrail
      Contact( #SysDI_Write.Ident_Instance.BUSY )
   END_RUNG wire#w1
   RUNG wire#powerrail
      Contact( #SysDI_Write.Ident_Instance.ERROR )
   END_RUNG wire#w1
   // the same network as SCL:
   IF #SysDI_Write.Ident_Instance.DONE OR #SysDI_Write.Ident_Instance.BUSY OR #SysDI_Write.Ident_Instance.ERROR THEN
       GOTO DiagSchreiben;
   END_IF;
END_REGION

REGION Network 20: HMI Diagnosis selection "End" / HMI-Diagnoseauswahl "Ende"
   RUNG wire#powerrail
      Contact( #t_VKE1 )
      JumpCoil( Ende )
   END_RUNG
   // the same network as SCL:
   IF #t_VKE1 THEN GOTO Ende; END_IF;
END_REGION

REGION Network 21: HMI Diagnosis Function Reset / HMI-Diagnose Funktion Reset
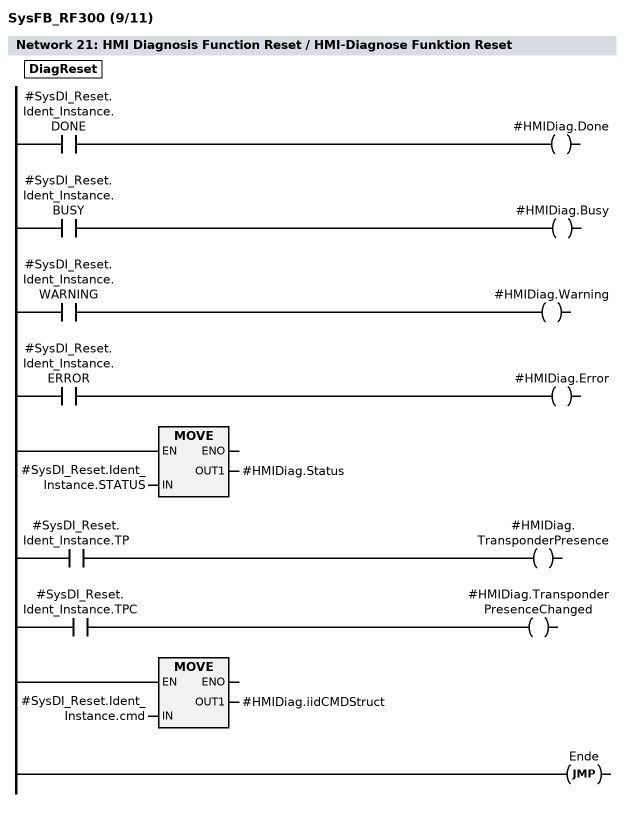
   Label( DiagReset )
   RUNG wire#powerrail
      Contact( #SysDI_Reset.Ident_Instance.DONE )
      Coil( #HMIDiag.Done )
   END_RUNG
   RUNG wire#powerrail
      Contact( #SysDI_Reset.Ident_Instance.BUSY )
      Coil( #HMIDiag.Busy )
   END_RUNG
   RUNG wire#powerrail
      Contact( #SysDI_Reset.Ident_Instance.WARNING )
      Coil( #HMIDiag.Warning )
   END_RUNG
   RUNG wire#powerrail
      Contact( #SysDI_Reset.Ident_Instance.ERROR )
      Coil( #HMIDiag.Error )
   END_RUNG
   RUNG wire#powerrail
      Move(in := #SysDI_Reset.Ident_Instance.STATUS, out1 => #HMIDiag.Status)
   END_RUNG
   RUNG wire#powerrail
      Contact( #SysDI_Reset.Ident_Instance.TP )
      Coil( #HMIDiag.TransponderPresence )
   END_RUNG
   RUNG wire#powerrail
      Contact( #SysDI_Reset.Ident_Instance.TPC )
      Coil( #HMIDiag.TransponderPresenceChanged )
   END_RUNG
   RUNG wire#powerrail
      Move(in := #SysDI_Reset.Ident_Instance.cmd, out1 => #HMIDiag.iidCMDStruct)
   END_RUNG
   RUNG wire#powerrail
      JumpCoil( Ende )
   END_RUNG
   // the same network as SCL:
   DiagReset:
   #HMIDiag.Done := #SysDI_Reset.Ident_Instance.DONE;
   #HMIDiag.Busy := #SysDI_Reset.Ident_Instance.BUSY;
   #HMIDiag.Warning := #SysDI_Reset.Ident_Instance.WARNING;
   #HMIDiag.Error := #SysDI_Reset.Ident_Instance.ERROR;
   #HMIDiag.Status := #SysDI_Reset.Ident_Instance.STATUS;
   #HMIDiag.TransponderPresence := #SysDI_Reset.Ident_Instance.TP;
   #HMIDiag.TransponderPresenceChanged := #SysDI_Reset.Ident_Instance.TPC;
   #HMIDiag.iidCMDStruct := #SysDI_Reset.Ident_Instance.cmd;
   GOTO Ende;
END_REGION

REGION Network 22: HMI Diagnosis Read function / HMI-Diagnose Funktion Lesen
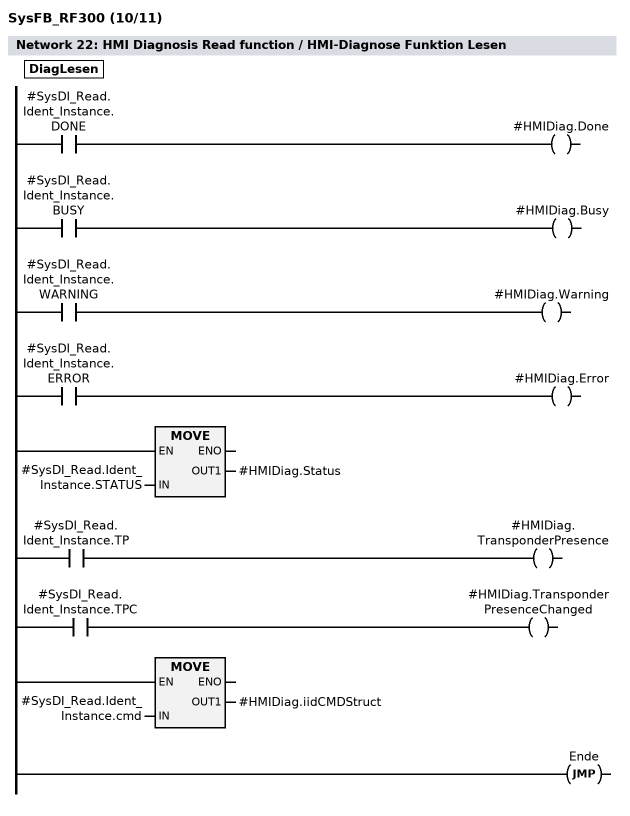
   Label( DiagLesen )
   RUNG wire#powerrail
      Contact( #SysDI_Read.Ident_Instance.DONE )
      Coil( #HMIDiag.Done )
   END_RUNG
   RUNG wire#powerrail
      Contact( #SysDI_Read.Ident_Instance.BUSY )
      Coil( #HMIDiag.Busy )
   END_RUNG
   RUNG wire#powerrail
      Contact( #SysDI_Read.Ident_Instance.WARNING )
      Coil( #HMIDiag.Warning )
   END_RUNG
   RUNG wire#powerrail
      Contact( #SysDI_Read.Ident_Instance.ERROR )
      Coil( #HMIDiag.Error )
   END_RUNG
   RUNG wire#powerrail
      Move(in := #SysDI_Read.Ident_Instance.STATUS, out1 => #HMIDiag.Status)
   END_RUNG
   RUNG wire#powerrail
      Contact( #SysDI_Read.Ident_Instance.TP )
      Coil( #HMIDiag.TransponderPresence )
   END_RUNG
   RUNG wire#powerrail
      Contact( #SysDI_Read.Ident_Instance.TPC )
      Coil( #HMIDiag.TransponderPresenceChanged )
   END_RUNG
   RUNG wire#powerrail
      Move(in := #SysDI_Read.Ident_Instance.cmd, out1 => #HMIDiag.iidCMDStruct)
   END_RUNG
   RUNG wire#powerrail
      JumpCoil( Ende )
   END_RUNG
   // the same network as SCL:
   DiagLesen:
   #HMIDiag.Done := #SysDI_Read.Ident_Instance.DONE;
   #HMIDiag.Busy := #SysDI_Read.Ident_Instance.BUSY;
   #HMIDiag.Warning := #SysDI_Read.Ident_Instance.WARNING;
   #HMIDiag.Error := #SysDI_Read.Ident_Instance.ERROR;
   #HMIDiag.Status := #SysDI_Read.Ident_Instance.STATUS;
   #HMIDiag.TransponderPresence := #SysDI_Read.Ident_Instance.TP;
   #HMIDiag.TransponderPresenceChanged := #SysDI_Read.Ident_Instance.TPC;
   #HMIDiag.iidCMDStruct := #SysDI_Read.Ident_Instance.cmd;
   GOTO Ende;
END_REGION

REGION Network 23: HMI Diagnosis Function Write / HMI-Diagnose Funktion Schreiben
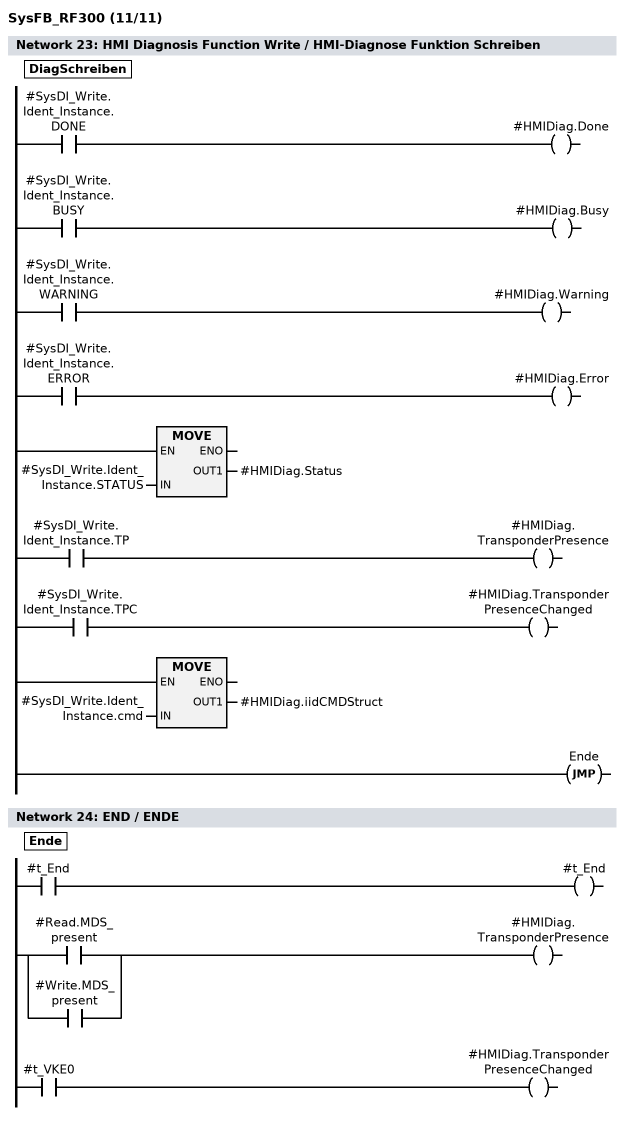
   Label( DiagSchreiben )
   RUNG wire#powerrail
      Contact( #SysDI_Write.Ident_Instance.DONE )
      Coil( #HMIDiag.Done )
   END_RUNG
   RUNG wire#powerrail
      Contact( #SysDI_Write.Ident_Instance.BUSY )
      Coil( #HMIDiag.Busy )
   END_RUNG
   RUNG wire#powerrail
      Contact( #SysDI_Write.Ident_Instance.WARNING )
      Coil( #HMIDiag.Warning )
   END_RUNG
   RUNG wire#powerrail
      Contact( #SysDI_Write.Ident_Instance.ERROR )
      Coil( #HMIDiag.Error )
   END_RUNG
   RUNG wire#powerrail
      Move(in := #SysDI_Write.Ident_Instance.STATUS, out1 => #HMIDiag.Status)
   END_RUNG
   RUNG wire#powerrail
      Contact( #SysDI_Write.Ident_Instance.TP )
      Coil( #HMIDiag.TransponderPresence )
   END_RUNG
   RUNG wire#powerrail
      Contact( #SysDI_Write.Ident_Instance.TPC )
      Coil( #HMIDiag.TransponderPresenceChanged )
   END_RUNG
   RUNG wire#powerrail
      Move(in := #SysDI_Write.Ident_Instance.cmd, out1 => #HMIDiag.iidCMDStruct)
   END_RUNG
   RUNG wire#powerrail
      JumpCoil( Ende )
   END_RUNG
   // the same network as SCL:
   DiagSchreiben:
   #HMIDiag.Done := #SysDI_Write.Ident_Instance.DONE;
   #HMIDiag.Busy := #SysDI_Write.Ident_Instance.BUSY;
   #HMIDiag.Warning := #SysDI_Write.Ident_Instance.WARNING;
   #HMIDiag.Error := #SysDI_Write.Ident_Instance.ERROR;
   #HMIDiag.Status := #SysDI_Write.Ident_Instance.STATUS;
   #HMIDiag.TransponderPresence := #SysDI_Write.Ident_Instance.TP;
   #HMIDiag.TransponderPresenceChanged := #SysDI_Write.Ident_Instance.TPC;
   #HMIDiag.iidCMDStruct := #SysDI_Write.Ident_Instance.cmd;
   GOTO Ende;
END_REGION

REGION Network 24: END / ENDE
   Label( Ende )
   RUNG wire#powerrail
      Contact( #t_End )
      Coil( #t_End )
   END_RUNG
   RUNG wire#powerrail
      Contact( #Read.MDS_present )
      wire#w1
      Coil( #HMIDiag.TransponderPresence )
   END_RUNG
   RUNG wire#powerrail
      Contact( #Write.MDS_present )
   END_RUNG wire#w1
   RUNG wire#powerrail
      Contact( #t_VKE0 )
      Coil( #HMIDiag.TransponderPresenceChanged )
   END_RUNG
   // the same network as SCL:
   Ende:
   #t_End := #t_End;
   #HMIDiag.TransponderPresence := #Read.MDS_present OR #Write.MDS_present;
   #HMIDiag.TransponderPresenceChanged := #t_VKE0;
END_REGION
END_FUNCTION_BLOCK
